(* IEC 61131-3 sources: CodesysTest/export/SX_1195.dev/Plc Logic/Application/PRJ Specific/Motion/Motors/Applied Motion/Applied Motion TSM34IP-3DG/Applied Motion TSM34IP-3DG Data Handlers/FB_StepServoFaultHandler.pou/FaultActive.prop, 1 file *)

(* ---- Get.pm.st ---- *)
(*#-#-#-#-#-#-#-#-#-#---Declaration---#-#-#-#-#-#-#-#-#-#-#-#-#*)

VAR
END_VAR
(*#-#-#-#-#-#-#-#-#-#---Implementation---#-#-#-#-#-#-#-#-#-#-#-#-#*)

FaultActive := faultCode <> 0;
